# B&R Automation Studio project BDD
Automation Studio 4.9

## Configuration Config1

CPU X90CP174.24-00, AutomationRuntime C4.90, Build 4.1.2, Vc V4.72.2

### Task classes (Cpu.sw)
```
Libraries: MpDatabase, MpBase, AsHttp, runtime
```

### Hardware
```
X90CP174_24_00 : X90CP174.24-00 v1.3.1.0  [X1 -> X1.SL]
  Module X1 (Type=X1, Virtual=true, Version=1.3.1.0)
    Connection (Connector=SL, TargetModule=X90CP174_24_00, TargetConnector=X1)
  Connector IF2:
    ActivateDevice = 1
  ConfigurationID = BDD_Config1
  Cyclic1Duration = 10000
  Cyclic1Tolerance = 10000
  Cyclic2Duration = 20000
  Cyclic2Tolerance = 20000
  Cyclic3Duration = 50000
  Cyclic3Tolerance = 50000
  Cyclic4Duration = 100000
  Cyclic4Tolerance = 100000
  Cyclic5Duration = 200000
  Cyclic5Tolerance = 200000
  Cyclic6Duration = 500000
  Cyclic6Tolerance = 500000
  Cyclic7Duration = 1000000
  Cyclic7Tolerance = 1000000
  Cyclic8Duration = 10000
  Cyclic8Tolerance = 30000000
```

### Config.mpdatabasecore - X90CP174_24_00/mappServices/Config.mpdatabasecore
```
Element gDatabaseCore (Type=mpdatabasecore)
  mapp.Database.Core:
    Name = BDDManitou
    UserName = Admin
    Password = Wiener_Blut27
    PortNumber = 3308
Element gDatabaseCore_1 (Type=mpdatabasecore)
```

## Logical view

Binary libraries used (declarations not repeated): MpDatabase, MpBase, AsHttp

### Program Logical/MDatabase (IEC)

#### Variables.var - Local variables
```iecst
VAR
	MpDatabaseCore_0 : USINT;
END_VAR
```

#### Cyclic.ld
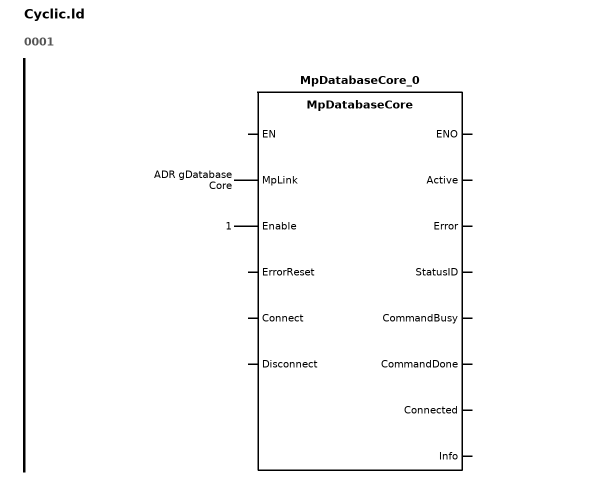
Ladder, written as Structured Text:
```iecst
PROGRAM _CYCLIC
(* Network 1 *)
MpDatabaseCore_0(MpLink := ADR(gDatabaseCore), Enable := 1);
END_PROGRAM
```

#### Exit.ld
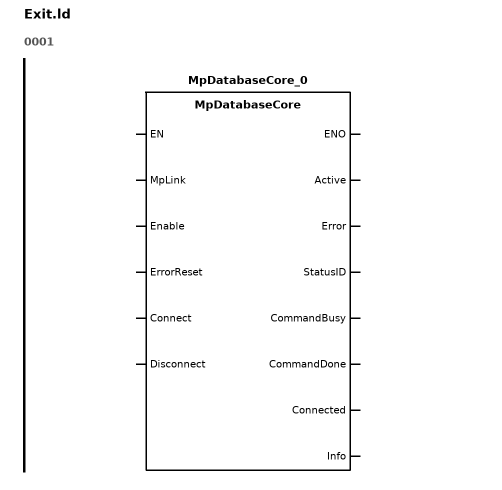
Ladder, written as Structured Text:
```iecst
PROGRAM _EXIT
(* Network 1 *)
MpDatabaseCore_0();
END_PROGRAM
```

#### Init.ld
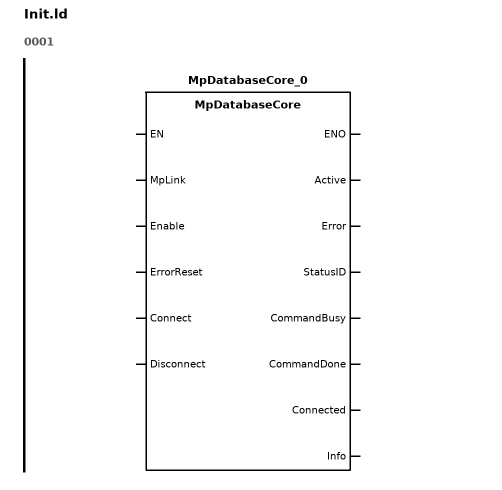
Ladder, written as Structured Text:
```iecst
PROGRAM _INIT
(* Network 1 *)
MpDatabaseCore_0();
END_PROGRAM
```

Listed in the project but not available here: Logical/Global.typ, Logical/Global.var, Logical/Libraries, Logical/MDatabase/Types.typ
